{attribute 'GeneratedUsingTerminal: EL9576-0000-0016'}
{attribute addProperty BoxType "EL9576-0000-0016"}
{attribute addProperty Id "Terminal_OvertemperatureAT %I*BOOL1I2T_errorAT %I*BOOL1I2T_warningAT %I*BOOL1OvervoltageAT %I*BOOL1UndervoltageAT %I*BOOL1Chopper_onAT %I*BOOL1DC_link_voltageAT %I*UDINT4Resistor_currentAT %I*DINT4Duty_cylceAT %I*USINT1"}
{attribute addProperty CRC "683767820"}
{attribute addProperty Size "15"}
TYPE BCT_Inputs_28C1780C :
STRUCT
	{attribute addProperty Name "Terminal_Overtemperature"}
	Terminal_Overtemperature AT %I* : BOOL;
	{attribute addProperty Name "I2T_error"}
	I2T_error AT %I* : BOOL;
	{attribute addProperty Name "I2T_warning"}
	I2T_warning AT %I* : BOOL;
	{attribute addProperty Name "Overvoltage"}
	Overvoltage AT %I* : BOOL;
	{attribute addProperty Name "Undervoltage"}
	Undervoltage AT %I* : BOOL;
	{attribute addProperty Name "Chopper_on"}
	Chopper_on AT %I* : BOOL;
	{attribute addProperty Name "DC_link_voltage"}
	DC_link_voltage AT %I* : UDINT;
	{attribute addProperty Name "Resistor_current"}
	Resistor_current AT %I* : DINT;
	{attribute addProperty Name "Duty_cylce"}
	Duty_cylce AT %I* : USINT;
END_STRUCT
END_TYPE

(* stored: Version 1.2.0.0, ProductVersion 3.1.4024.9
   DUT BCT_Inputs_28C1780C: Id {76ae642b-159b-4a76-ac0d-84cf51e40f35} *)
